Fanuc KAREL source: kb00045.KL

-- PROVISIONAL review KL for V770-1; original PC SHA256 2ea1711d99bf3b58d467f98c2392068af86bae187434bae2a8597f10d2b0d95a
-- Incomplete behavior may be omitted. Consult companion uncertainty JSON. Do not deploy.
PROGRAM KB00045
%NOLOCKGROUP
BEGIN
  -- UNRESOLVED_PC offsets 5-14; opcodes 3F,75
  -- UNRESOLVED_PC offsets 19-26; opcodes 9D,23
  -- UNRESOLVED_PC offsets 31-49; opcodes 27,22,2A,22,31
  -- UNRESOLVED_PC offsets 54-58; opcodes 7F
END KB00045
